(* Logix 5000 project; controller R5_CSS vendor 1 type 14 code 74 rev 19.11; software revision 19.01; part 14 of 20 *)
(* tags used below, declared in another part *)
   CSS_Heartbeat : BOOL;
   CSS_OK_TO_RUN : BOOL;   // PRU_RUN_DISABLE 0 = Cannot Run 1 = OK to Run
   CSS_OK_TO_START : BOOL;   // PRU_START_DISABLE 0 = Cannot Start 1 = OK to Start
   HS104A : ValveControl_TwoWay;
   HS104B : ValveControl_TwoWay;
   LC101 : LEVEL_CONTROL;   // QUENCH TOWER BASIN LIT
   LC303A : LEVEL_CONTROL;   // AQUEOUS PHASE OF PRIMARY SETTLER
   ONE_SHOT : BOOL[32];
   ONE_SHOT_P101B : BOOL;
   P101A : PUMP_CONTROL;
   P101A_BumpStartONS : BOOL;
   P101A_QI_AUTO_OS : BOOL;
   P101A_QI_MAN_OS : BOOL;
   P101B : PUMP_CONTROL;
   P101B_BumpStartONS : BOOL;
   P101B_QI_AUTO_OS : BOOL;
   P101B_QI_MAN_OS : BOOL;
   PRU_BLOWER_SEQ : INT;   // PRU BLOWER SEQUENCE NUMBER
   PRU_DELAY_REQ : INT;
   PRU_MaxTempDelayMin : REAL;
   PRU_MaxTempDelta : REAL;
   PRU_PT404 : REAL[10];
   PRU_PT404_Done : REAL[10];
   PRU_PT404_Max : REAL[10];
   PRU_RECIPE_LOAD : INT;
   PRU_RECIPE_LOAD_DLY : TIMER[10];
   PRU_RunDoneTemp : BOOL[32];
   PRU_RunDoneTime : BOOL[32];
   PRU_Running : BOOL[32];
   PRU_RunningMaxHrs : REAL;
   PRU_RunningMaxTempDelay : TIMER[10];
   PRU_RunningMinutePulse : TIMER[10];
   PRU_RunningTotalMin : COUNTER[10];
   PRU_START_REQ : INT;
   PRUD_CHANGE : INT;
   PRUD_CHANGE_OF_STATE : BOOL;
   PRUD_COMMS_TIMER : TIMER;
   PRUD_ECOOL : BOOL;
   PRUD_ECOOL_TON : TIMER;
   PRUD_HeartbeatCommsLoss : BOOL;
   PRUD_HeartbeatOffONS : BOOL;
   PRUD_HeartbeatOnONS : BOOL;
   PRUD_READ : INT[30];   // PRU D READ
   PRUD_START_REQ_ONS : BOOL[32];
   PRUD_WRITE : INT[40];
   TC101A : TEMP_CONTROL;   // QUENCH BASIN TRANSFER BASIN A TEMPERATURE CONTROL
   TC101B : TEMP_CONTROL;   // QUENCH BASIN TRANSFER BASIN B TEMPERATURE CONTROL
   TIMER : TIMER[50];   // HX A TIMER FOR START
   UTL_Comms : DINT[3];
   UTL_CommsLossAlm : BOOL;
(* MainProgram, continued *)

ROUTINE PRUD   (* ladder *)
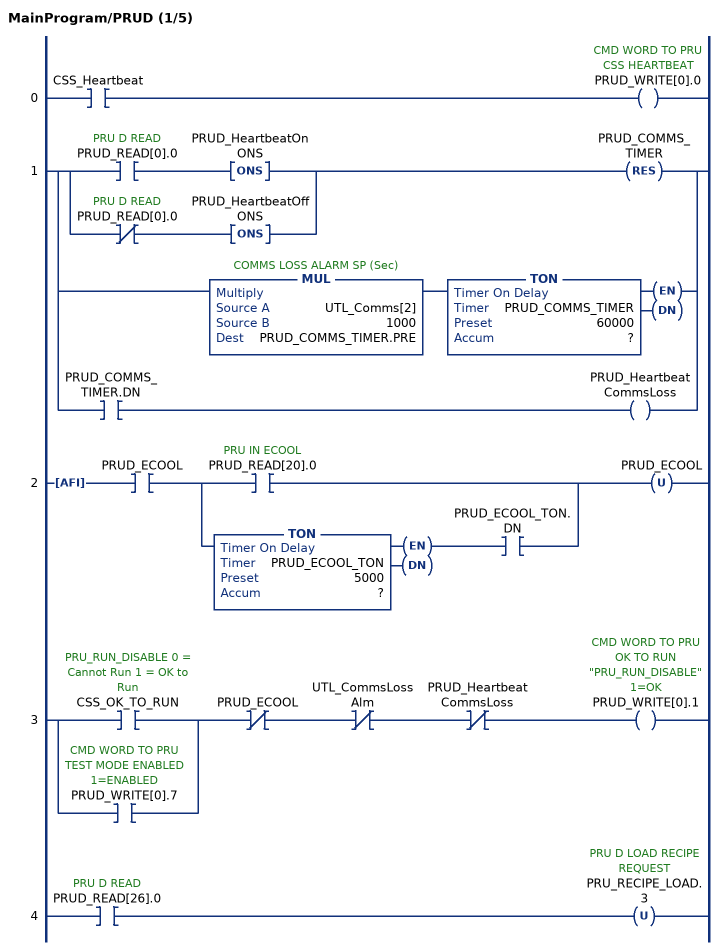
   0: XIC(CSS_Heartbeat)OTE(PRUD_WRITE[0].0);
   1: [[XIC(PRUD_READ[0].0) ONS(PRUD_HeartbeatOnONS) ,XIO(PRUD_READ[0].0) ONS(PRUD_HeartbeatOffONS) ] RES(PRUD_COMMS_TIMER) ,MUL(UTL_Comms[2],1000,PRUD_COMMS_TIMER.PRE) TON(PRUD_COMMS_TIMER,?,?) ,XIC(PRUD_COMMS_TIMER.DN) OTE(PRUD_HeartbeatCommsLoss) ];
   2: AFI()XIC(PRUD_ECOOL)[XIC(PRUD_READ[20].0) ,TON(PRUD_ECOOL_TON,?,?) XIC(PRUD_ECOOL_TON.DN) ]OTU(PRUD_ECOOL);
   3: [XIC(CSS_OK_TO_RUN) ,XIC(PRUD_WRITE[0].7) ]XIO(PRUD_ECOOL)XIO(UTL_CommsLossAlm)XIO(PRUD_HeartbeatCommsLoss)OTE(PRUD_WRITE[0].1);
   4: XIC(PRUD_READ[26].0)OTU(PRU_RECIPE_LOAD.3);
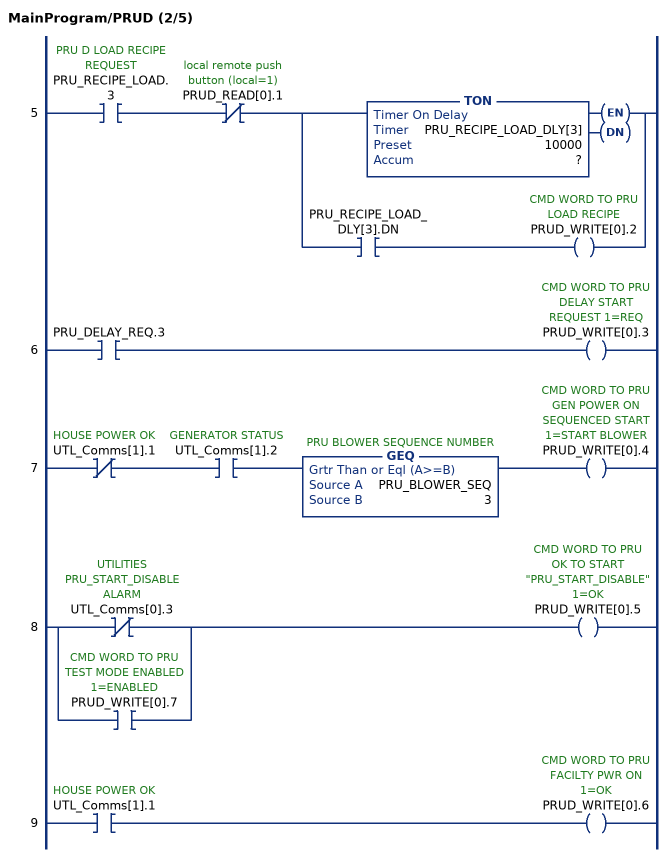
   5: XIC(PRU_RECIPE_LOAD.3)XIO(PRUD_READ[0].1)[TON(PRU_RECIPE_LOAD_DLY[3],?,?) ,XIC(PRU_RECIPE_LOAD_DLY[3].DN) OTE(PRUD_WRITE[0].2) ];
   6: XIC(PRU_DELAY_REQ.3)OTE(PRUD_WRITE[0].3);
   7: XIO(UTL_Comms[1].1)XIC(UTL_Comms[1].2)GEQ(PRU_BLOWER_SEQ,3)OTE(PRUD_WRITE[0].4);
   8: [XIO(UTL_Comms[0].3) ,XIC(PRUD_WRITE[0].7) ]OTE(PRUD_WRITE[0].5);
   9: XIC(UTL_Comms[1].1)OTE(PRUD_WRITE[0].6);
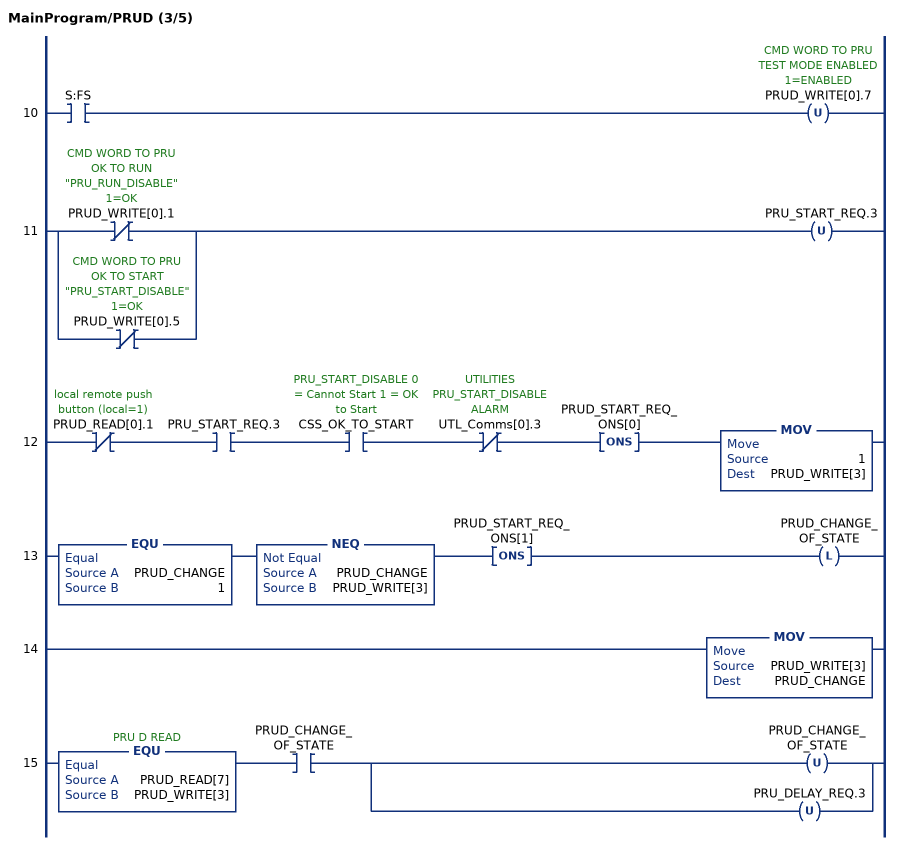
   10: XIC(S:FS)OTU(PRUD_WRITE[0].7);
   11: [XIO(PRUD_WRITE[0].1) ,XIO(PRUD_WRITE[0].5) ]OTU(PRU_START_REQ.3);
   12: XIO(PRUD_READ[0].1)XIC(PRU_START_REQ.3)XIC(CSS_OK_TO_START)XIO(UTL_Comms[0].3)ONS(PRUD_START_REQ_ONS[0])MOV(1,PRUD_WRITE[3]);
   13: EQU(PRUD_CHANGE,1)NEQ(PRUD_CHANGE,PRUD_WRITE[3])ONS(PRUD_START_REQ_ONS[1])OTL(PRUD_CHANGE_OF_STATE);
   14: MOV(PRUD_WRITE[3],PRUD_CHANGE);
   15: EQU(PRUD_READ[7],PRUD_WRITE[3])XIC(PRUD_CHANGE_OF_STATE)[OTU(PRUD_CHANGE_OF_STATE) ,OTU(PRU_DELAY_REQ.3) ];
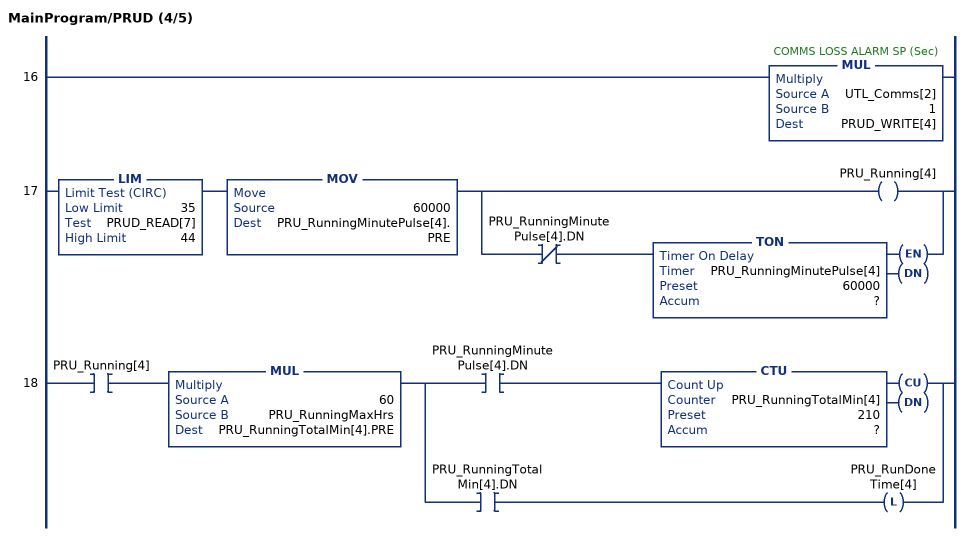
   16: MUL(UTL_Comms[2],1,PRUD_WRITE[4]);
   17: LIM(35,PRUD_READ[7],44)MOV(60000,PRU_RunningMinutePulse[4].PRE)[OTE(PRU_Running[4]) ,XIO(PRU_RunningMinutePulse[4].DN) TON(PRU_RunningMinutePulse[4],?,?) ];
   18: XIC(PRU_Running[4])MUL(60,PRU_RunningMaxHrs,PRU_RunningTotalMin[4].PRE)[XIC(PRU_RunningMinutePulse[4].DN) CTU(PRU_RunningTotalMin[4],?,?) ,XIC(PRU_RunningTotalMin[4].DN) OTL(PRU_RunDoneTime[4]) ];
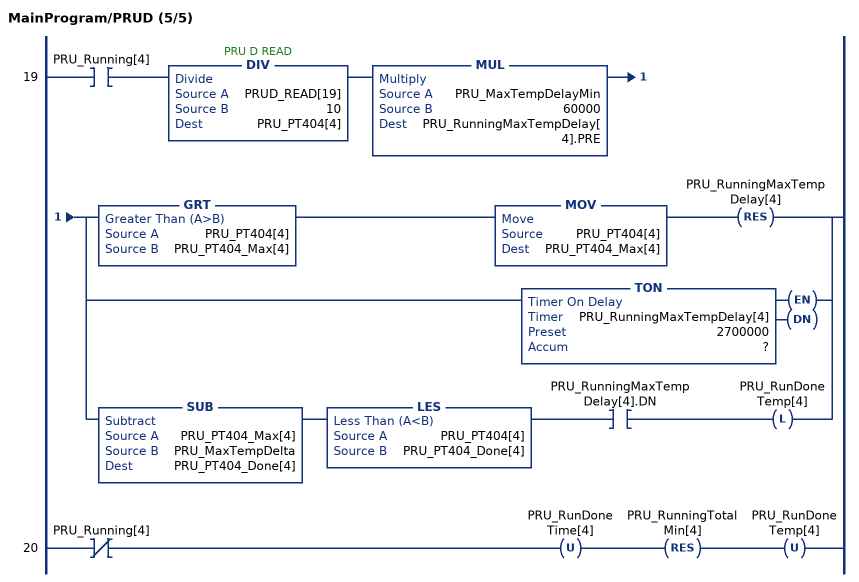
   19: XIC(PRU_Running[4])DIV(PRUD_READ[19],10,PRU_PT404[4])MUL(PRU_MaxTempDelayMin,60000,PRU_RunningMaxTempDelay[4].PRE)[GRT(PRU_PT404[4],PRU_PT404_Max[4]) MOV(PRU_PT404[4],PRU_PT404_Max[4]) RES(PRU_RunningMaxTempDelay[4]) ,TON(PRU_RunningMaxTempDelay[4],?,?) ,SUB(PRU_PT404_Max[4],PRU_MaxTempDelta,PRU_PT404_Done[4]) LES(PRU_PT404[4],PRU_PT404_Done[4]) XIC(PRU_RunningMaxTempDelay[4].DN) OTL(PRU_RunDoneTemp[4]) ];
   20: XIO(PRU_Running[4])OTU(PRU_RunDoneTime[4])RES(PRU_RunningTotalMin[4])OTU(PRU_RunDoneTemp[4]);
END_ROUTINE

ROUTINE Pump101A_BasinPumpControl   (* ladder *)
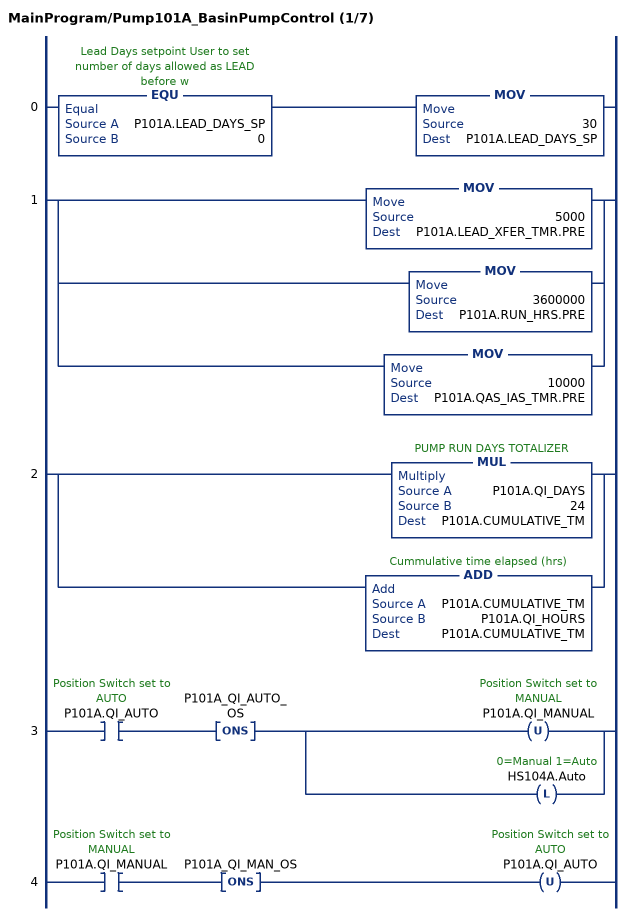
   0: EQU(P101A.LEAD_DAYS_SP,0)MOV(30,P101A.LEAD_DAYS_SP);
   1: [MOV(5000,P101A.LEAD_XFER_TMR.PRE) ,MOV(3600000,P101A.RUN_HRS.PRE) ,MOV(10000,P101A.QAS_IAS_TMR.PRE) ];
   2: [MUL(P101A.QI_DAYS,24,P101A.CUMULATIVE_TM) ,ADD(P101A.CUMULATIVE_TM,P101A.QI_HOURS,P101A.CUMULATIVE_TM) ];
   3: XIC(P101A.QI_AUTO)ONS(P101A_QI_AUTO_OS)[OTU(P101A.QI_MANUAL) ,OTL(HS104A.Auto) ];
   4: XIC(P101A.QI_MANUAL)ONS(P101A_QI_MAN_OS)OTU(P101A.QI_AUTO);
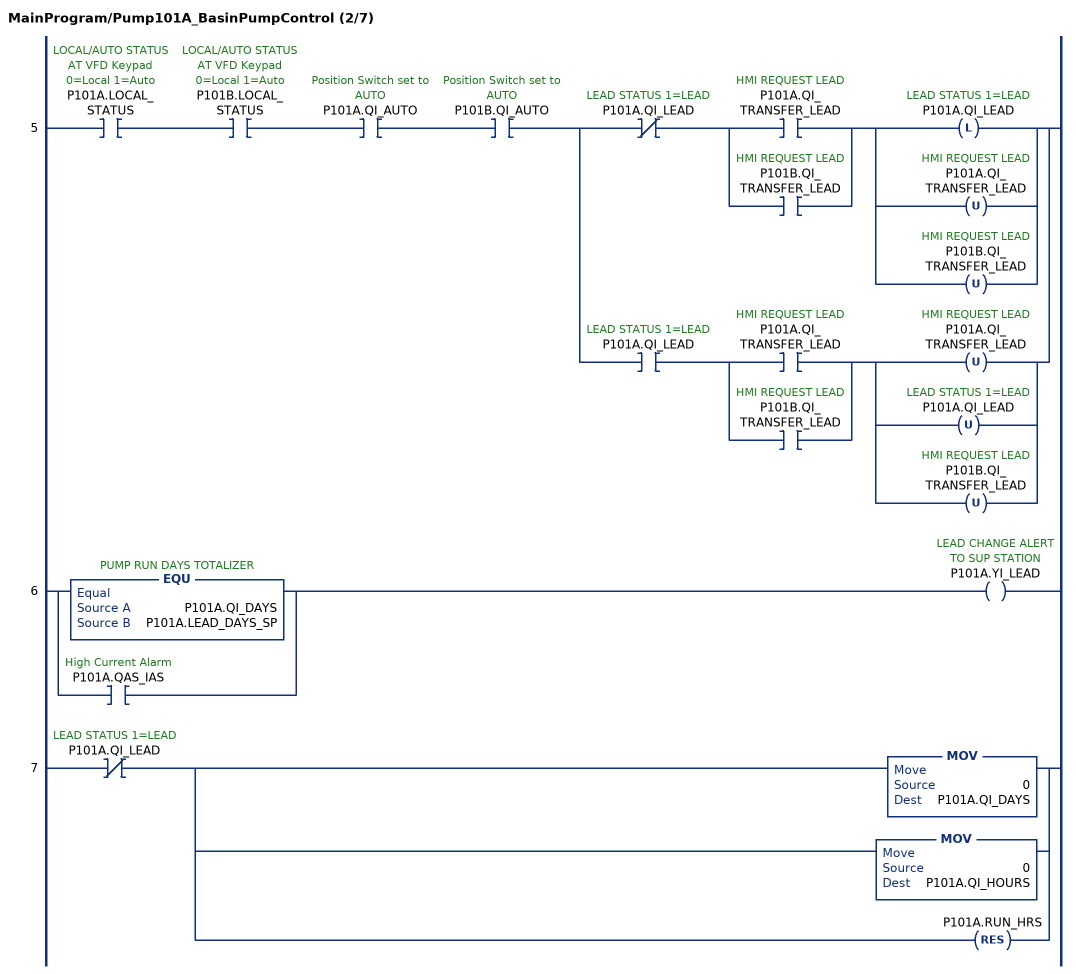
   5: XIC(P101A.LOCAL_STATUS)XIC(P101B.LOCAL_STATUS)XIC(P101A.QI_AUTO)XIC(P101B.QI_AUTO)[XIO(P101A.QI_LEAD) [XIC(P101A.QI_TRANSFER_LEAD) ,XIC(P101B.QI_TRANSFER_LEAD) ] [OTL(P101A.QI_LEAD) ,OTU(P101A.QI_TRANSFER_LEAD) ,OTU(P101B.QI_TRANSFER_LEAD) ] ,XIC(P101A.QI_LEAD) [XIC(P101A.QI_TRANSFER_LEAD) ,XIC(P101B.QI_TRANSFER_LEAD) ] [OTU(P101A.QI_TRANSFER_LEAD) ,OTU(P101A.QI_LEAD) ,OTU(P101B.QI_TRANSFER_LEAD) ] ];
   6: [EQU(P101A.QI_DAYS,P101A.LEAD_DAYS_SP) ,XIC(P101A.QAS_IAS) ]OTE(P101A.YI_LEAD);
   7: XIO(P101A.QI_LEAD)[MOV(0,P101A.QI_DAYS) ,MOV(0,P101A.QI_HOURS) ,RES(P101A.RUN_HRS) ];
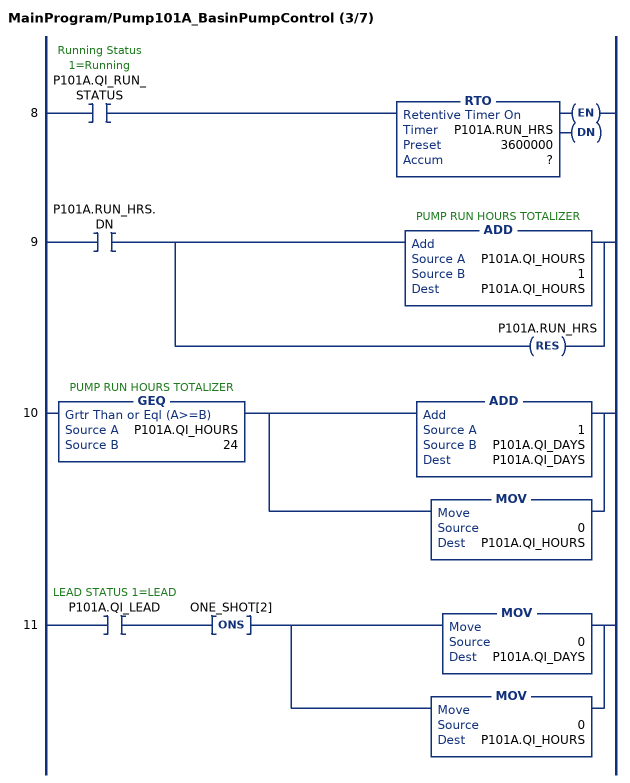
   8: XIC(P101A.QI_RUN_STATUS)RTO(P101A.RUN_HRS,?,?);
   9: XIC(P101A.RUN_HRS.DN)[ADD(P101A.QI_HOURS,1,P101A.QI_HOURS) ,RES(P101A.RUN_HRS) ];
   10: GEQ(P101A.QI_HOURS,24)[ADD(1,P101A.QI_DAYS,P101A.QI_DAYS) ,MOV(0,P101A.QI_HOURS) ];
   11: XIC(P101A.QI_LEAD)ONS(ONE_SHOT[2])[MOV(0,P101A.QI_DAYS) ,MOV(0,P101A.QI_HOURS) ];
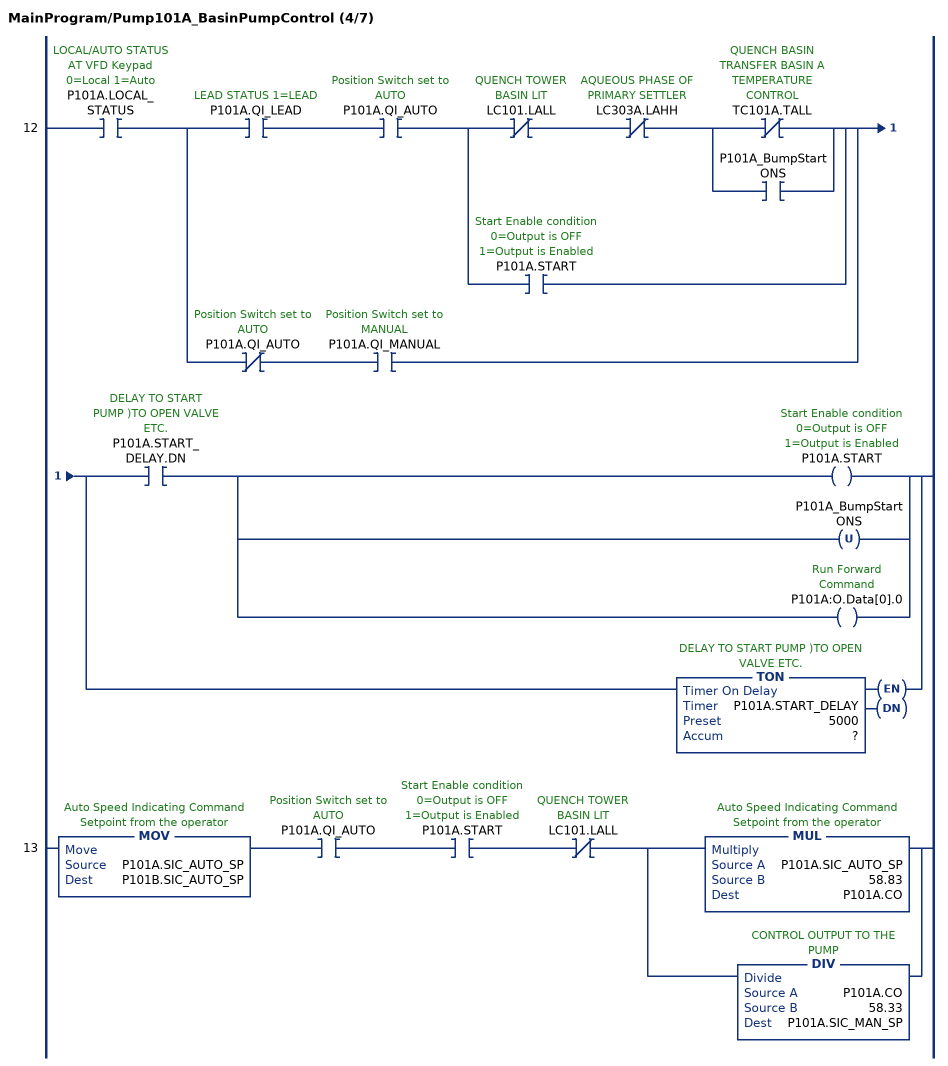
   12: XIC(P101A.LOCAL_STATUS)[XIC(P101A.QI_LEAD) XIC(P101A.QI_AUTO) [XIO(LC101.LALL) XIO(LC303A.LAHH) [XIO(TC101A.TALL) ,XIC(P101A_BumpStartONS) ] ,XIC(P101A.START) ] ,XIO(P101A.QI_AUTO) XIC(P101A.QI_MANUAL) ][XIC(P101A.START_DELAY.DN) [OTE(P101A.START) ,OTU(P101A_BumpStartONS) ,OTE(P101A:O.Data[0].0) ] ,TON(P101A.START_DELAY,?,?) ];
   13: MOV(P101A.SIC_AUTO_SP,P101B.SIC_AUTO_SP)XIC(P101A.QI_AUTO)XIC(P101A.START)XIO(LC101.LALL)[MUL(P101A.SIC_AUTO_SP,58.83,P101A.CO) ,DIV(P101A.CO,58.33,P101A.SIC_MAN_SP) ];
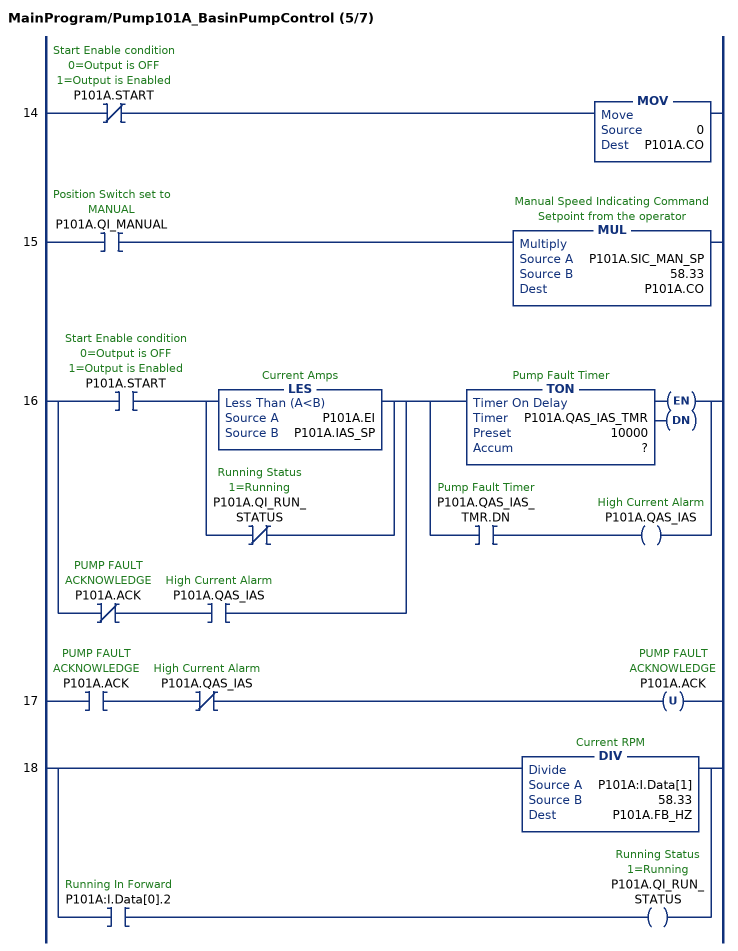
   14: XIO(P101A.START)MOV(0,P101A.CO);
   15: XIC(P101A.QI_MANUAL)MUL(P101A.SIC_MAN_SP,58.33,P101A.CO);
   16: [XIC(P101A.START) [LES(P101A.EI,P101A.IAS_SP) ,XIO(P101A.QI_RUN_STATUS) ] ,XIO(P101A.ACK) XIC(P101A.QAS_IAS) ][TON(P101A.QAS_IAS_TMR,?,?) ,XIC(P101A.QAS_IAS_TMR.DN) OTE(P101A.QAS_IAS) ];
   17: XIC(P101A.ACK)XIO(P101A.QAS_IAS)OTU(P101A.ACK);
   18: [DIV(P101A:I.Data[1],58.33,P101A.FB_HZ) ,XIC(P101A:I.Data[0].2) OTE(P101A.QI_RUN_STATUS) ];
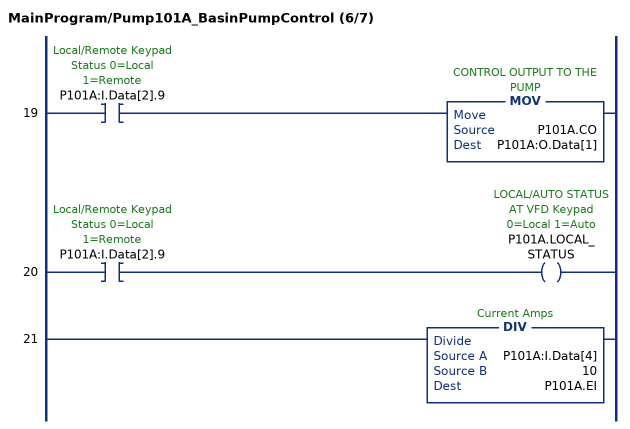
   19: XIC(P101A:I.Data[2].9)MOV(P101A.CO,P101A:O.Data[1]);
   20: XIC(P101A:I.Data[2].9)OTE(P101A.LOCAL_STATUS);
   21: DIV(P101A:I.Data[4],10,P101A.EI);
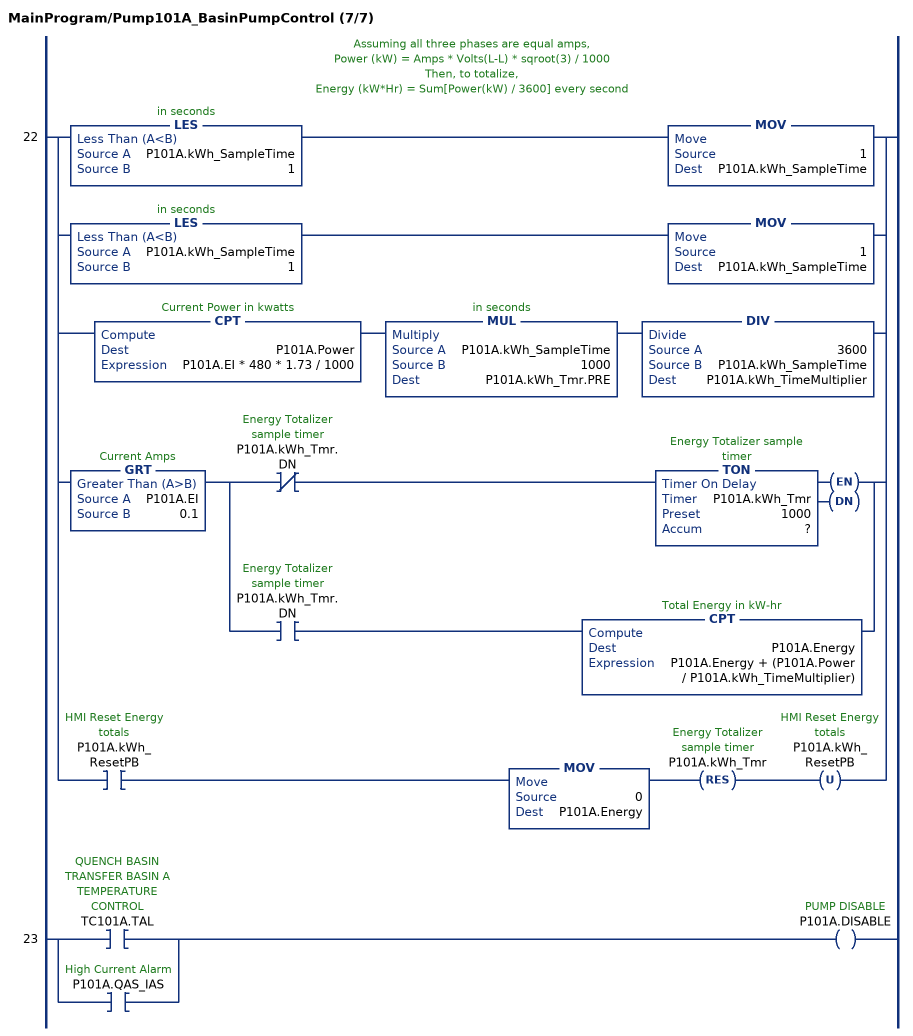
   // Assuming all three phases are equal amps,
   // Power (kW) = Amps * Volts(L-L) * sqroot(3) / 1000
   // Then, to totalize,
   // Energy (kW*Hr) = Sum[Power(kW) / 3600] every second
   22: [[LES(P101A.kWh_SampleTime,1) MOV(1,P101A.kWh_SampleTime) ,LES(P101A.kWh_SampleTime,1) MOV(1,P101A.kWh_SampleTime) ] ,CPT(P101A.Power,P101A.EI * 480 * 1.73 / 1000) MUL(P101A.kWh_SampleTime,1000,P101A.kWh_Tmr.PRE) DIV(3600,P101A.kWh_SampleTime,P101A.kWh_TimeMultiplier) ,GRT(P101A.EI,0.1) [XIO(P101A.kWh_Tmr.DN) TON(P101A.kWh_Tmr,?,?) ,XIC(P101A.kWh_Tmr.DN) CPT(P101A.Energy,P101A.Energy + (P101A.Power / P101A.kWh_TimeMultiplier)) ] ,XIC(P101A.kWh_ResetPB) MOV(0,P101A.Energy) RES(P101A.kWh_Tmr) OTU(P101A.kWh_ResetPB) ];
   23: [XIC(TC101A.TAL) ,XIC(P101A.QAS_IAS) ]OTE(P101A.DISABLE);
END_ROUTINE

ROUTINE Pump101B_BasinPumpControl   (* ladder *)
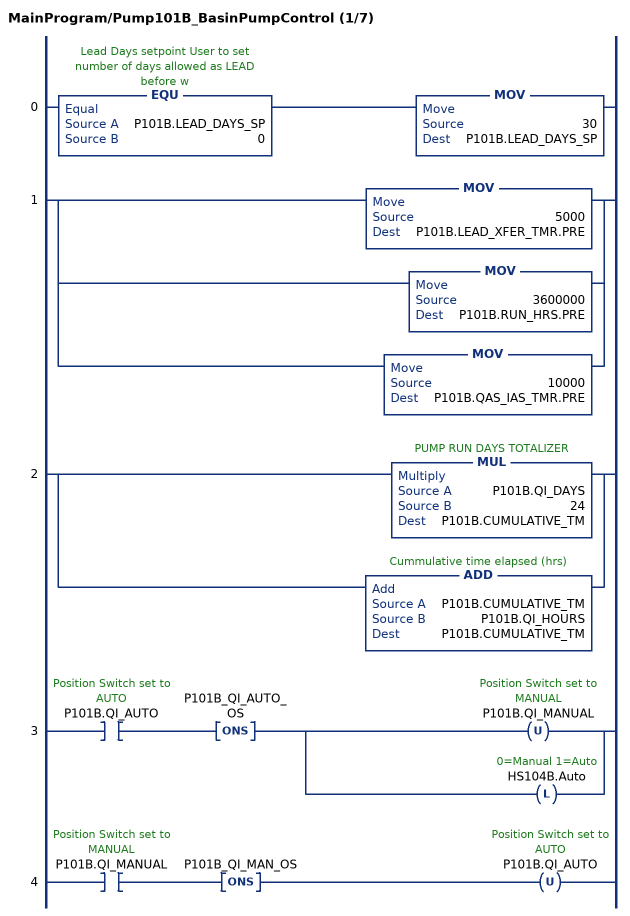
   0: EQU(P101B.LEAD_DAYS_SP,0)MOV(30,P101B.LEAD_DAYS_SP);
   1: [MOV(5000,P101B.LEAD_XFER_TMR.PRE) ,MOV(3600000,P101B.RUN_HRS.PRE) ,MOV(10000,P101B.QAS_IAS_TMR.PRE) ];
   2: [MUL(P101B.QI_DAYS,24,P101B.CUMULATIVE_TM) ,ADD(P101B.CUMULATIVE_TM,P101B.QI_HOURS,P101B.CUMULATIVE_TM) ];
   3: XIC(P101B.QI_AUTO)ONS(P101B_QI_AUTO_OS)[OTU(P101B.QI_MANUAL) ,OTL(HS104B.Auto) ];
   4: XIC(P101B.QI_MANUAL)ONS(P101B_QI_MAN_OS)OTU(P101B.QI_AUTO);
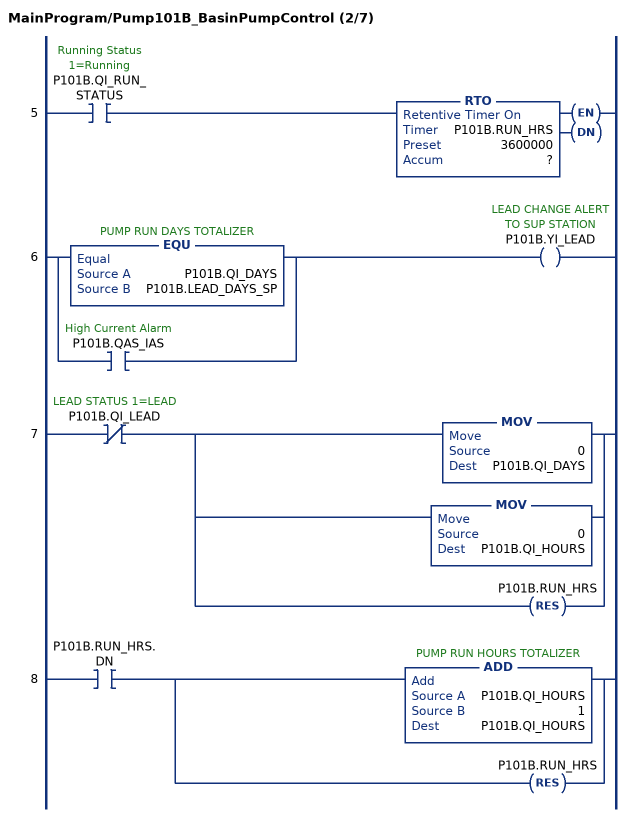
   5: XIC(P101B.QI_RUN_STATUS)RTO(P101B.RUN_HRS,?,?);
   6: [EQU(P101B.QI_DAYS,P101B.LEAD_DAYS_SP) ,XIC(P101B.QAS_IAS) ]OTE(P101B.YI_LEAD);
   7: XIO(P101B.QI_LEAD)[MOV(0,P101B.QI_DAYS) ,MOV(0,P101B.QI_HOURS) ,RES(P101B.RUN_HRS) ];
   8: XIC(P101B.RUN_HRS.DN)[ADD(P101B.QI_HOURS,1,P101B.QI_HOURS) ,RES(P101B.RUN_HRS) ];
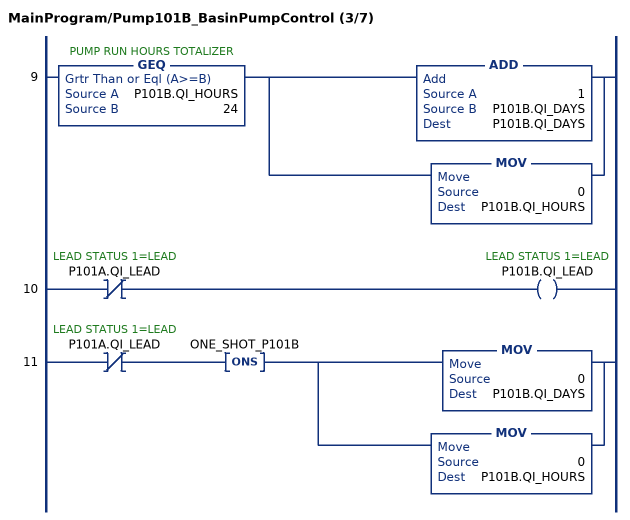
   9: GEQ(P101B.QI_HOURS,24)[ADD(1,P101B.QI_DAYS,P101B.QI_DAYS) ,MOV(0,P101B.QI_HOURS) ];
   10: XIO(P101A.QI_LEAD)OTE(P101B.QI_LEAD);
   11: XIO(P101A.QI_LEAD)ONS(ONE_SHOT_P101B)[MOV(0,P101B.QI_DAYS) ,MOV(0,P101B.QI_HOURS) ];
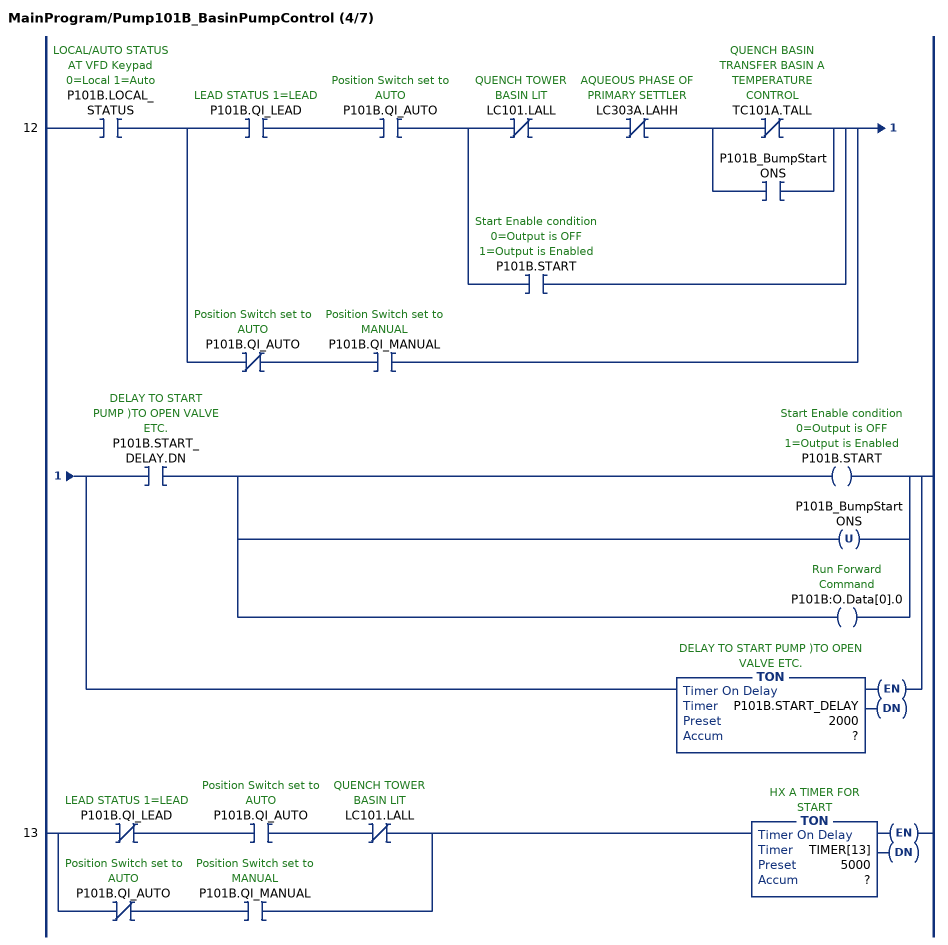
   12: XIC(P101B.LOCAL_STATUS)[XIC(P101B.QI_LEAD) XIC(P101B.QI_AUTO) [XIO(LC101.LALL) XIO(LC303A.LAHH) [XIO(TC101A.TALL) ,XIC(P101B_BumpStartONS) ] ,XIC(P101B.START) ] ,XIO(P101B.QI_AUTO) XIC(P101B.QI_MANUAL) ][XIC(P101B.START_DELAY.DN) [OTE(P101B.START) ,OTU(P101B_BumpStartONS) ,OTE(P101B:O.Data[0].0) ] ,TON(P101B.START_DELAY,?,?) ];
   13: [XIO(P101B.QI_LEAD) XIC(P101B.QI_AUTO) XIO(LC101.LALL) ,XIO(P101B.QI_AUTO) XIC(P101B.QI_MANUAL) ]TON(TIMER[13],?,?);
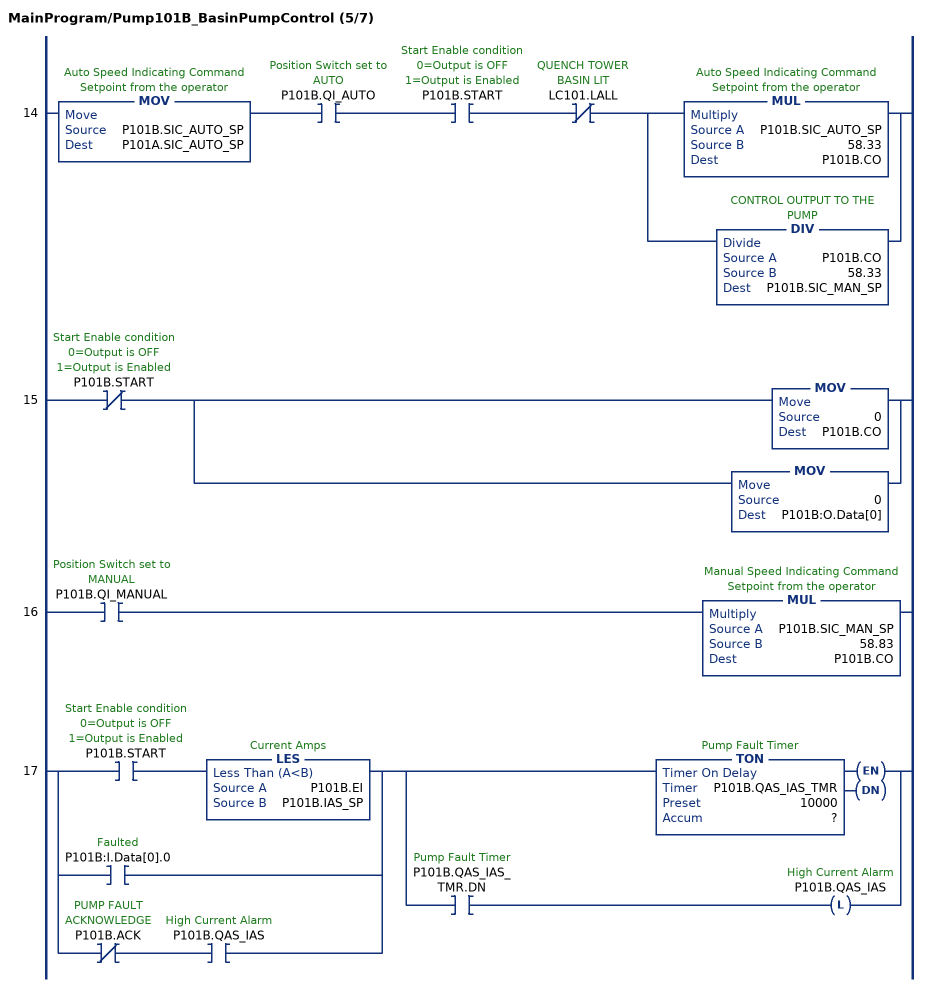
   14: MOV(P101B.SIC_AUTO_SP,P101A.SIC_AUTO_SP)XIC(P101B.QI_AUTO)XIC(P101B.START)XIO(LC101.LALL)[MUL(P101B.SIC_AUTO_SP,58.33,P101B.CO) ,DIV(P101B.CO,58.33,P101B.SIC_MAN_SP) ];
   15: XIO(P101B.START)[MOV(0,P101B.CO) ,MOV(0,P101B:O.Data[0]) ];
   16: XIC(P101B.QI_MANUAL)MUL(P101B.SIC_MAN_SP,58.83,P101B.CO);
   17: [XIC(P101B.START) LES(P101B.EI,P101B.IAS_SP) ,XIC(P101B:I.Data[0].0) ,XIO(P101B.ACK) XIC(P101B.QAS_IAS) ][TON(P101B.QAS_IAS_TMR,?,?) ,XIC(P101B.QAS_IAS_TMR.DN) OTL(P101B.QAS_IAS) ];
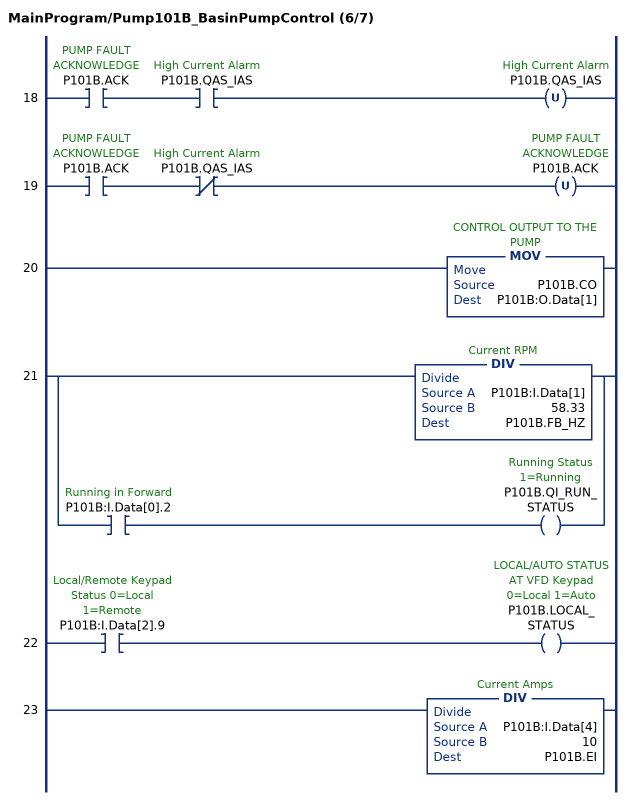
   18: XIC(P101B.ACK)XIC(P101B.QAS_IAS)OTU(P101B.QAS_IAS);
   19: XIC(P101B.ACK)XIO(P101B.QAS_IAS)OTU(P101B.ACK);
   20: MOV(P101B.CO,P101B:O.Data[1]);
   21: [DIV(P101B:I.Data[1],58.33,P101B.FB_HZ) ,XIC(P101B:I.Data[0].2) OTE(P101B.QI_RUN_STATUS) ];
   22: XIC(P101B:I.Data[2].9)OTE(P101B.LOCAL_STATUS);
   23: DIV(P101B:I.Data[4],10,P101B.EI);
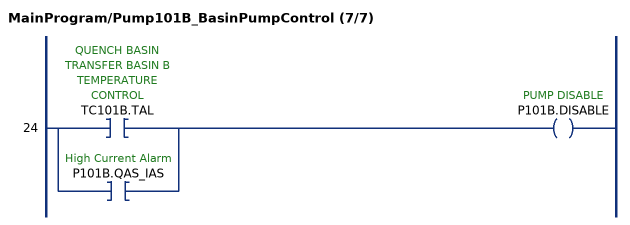
   24: [XIC(TC101B.TAL) ,XIC(P101B.QAS_IAS) ]OTE(P101B.DISABLE);
END_ROUTINE
